// TIA Portal V15.1 export
// export: Created 2019-08-01T08:30:35.1738307Z, ExportSetting None, DisplayName Totally Integrated Automation Portal, DisplayVersion V15.1, DisplayName TIA Portal Openness, DisplayVersion V15.1, DisplayName STEP 7 Professional, DisplayVersion V15.1, DisplayName STEP 7 Safety, DisplayVersion V15.1, DisplayName WinCC Advanced, DisplayVersion V15.1
TYPE "type#SKILL_NAME#GetResultParameter_Out"
END_TYPE
